{attribute addProperty BoxType "EPP6228-0022-0016"}
{attribute addProperty Id "DeviceState_InputsDeviceState_Inputs_DB789D68648"}
{attribute addProperty CRC "3967119980"}
{attribute addProperty SizeInBites "64"}
{attribute addProperty SizeInBytes "8"}
TYPE Module_2_DeviceState_Inputs_EC75726C :
STRUCT
	{attribute addProperty Name "DeviceState_Inputs"}
	DeviceState_Inputs  : DeviceState_Inputs_DB789D68;
END_STRUCT
END_TYPE

(* stored: Version 1.2.0.0, ProductVersion 3.1.4024.9
   DUT Module_2_DeviceState_Inputs_EC75726C: Id {b8b6ebc7-9b6e-46b5-97af-b928ce815754} *)
